// TIA Portal V19 export
FUNCTION "FC90_SentronComm" : Void   // FC90, LAD
{ S7_Optimized_Access := 'TRUE' }
// stored: AutoNumber false, IsIECCheckEnabled true, SetENOAutomatically false
BEGIN

REGION Network 1: Read Sentron Main cabinet
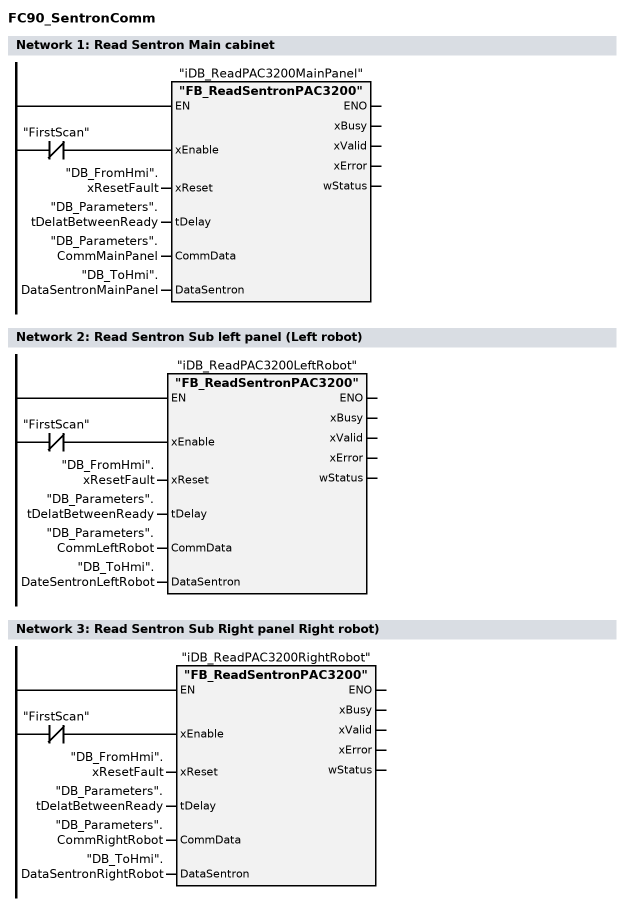
   RUNG wire#powerrail
      "iDB_ReadPAC3200MainPanel"(xEnable := wire#w1, xReset := "DB_FromHmi".xResetFault, tDelay := "DB_Parameters".tDelatBetweenReady, CommData := "DB_Parameters".CommMainPanel, DataSentron := "DB_ToHmi".DataSentronMainPanel, xBusy =>, xValid =>, xError =>, wStatus =>)
   END_RUNG
   RUNG wire#powerrail
      I_Contact( "FirstScan" )
   END_RUNG wire#w1
   // the same network as SCL:
   "iDB_ReadPAC3200MainPanel"(xEnable := NOT "FirstScan",   // "FB_ReadSentronPAC3200"
                           xReset := "DB_FromHmi".xResetFault,
                           tDelay := "DB_Parameters".tDelatBetweenReady,
                           CommData := "DB_Parameters".CommMainPanel,
                           DataSentron := "DB_ToHmi".DataSentronMainPanel);
END_REGION

REGION Network 2: Read Sentron Sub left panel (Left robot)
   RUNG wire#powerrail
      "iDB_ReadPAC3200LeftRobot"(xEnable := wire#w1, xReset := "DB_FromHmi".xResetFault, tDelay := "DB_Parameters".tDelatBetweenReady, CommData := "DB_Parameters".CommLeftRobot, DataSentron := "DB_ToHmi".DateSentronLeftRobot, xBusy =>, xValid =>, xError =>, wStatus =>)
   END_RUNG
   RUNG wire#powerrail
      I_Contact( "FirstScan" )
   END_RUNG wire#w1
   // the same network as SCL:
   "iDB_ReadPAC3200LeftRobot"(xEnable := NOT "FirstScan",   // "FB_ReadSentronPAC3200"
                           xReset := "DB_FromHmi".xResetFault,
                           tDelay := "DB_Parameters".tDelatBetweenReady,
                           CommData := "DB_Parameters".CommLeftRobot,
                           DataSentron := "DB_ToHmi".DateSentronLeftRobot);
END_REGION

REGION Network 3: Read Sentron Sub Right panel Right robot)
   RUNG wire#powerrail
      "iDB_ReadPAC3200RightRobot"(xEnable := wire#w1, xReset := "DB_FromHmi".xResetFault, tDelay := "DB_Parameters".tDelatBetweenReady, CommData := "DB_Parameters".CommRightRobot, DataSentron := "DB_ToHmi".DataSentronRightRobot, xBusy =>, xValid =>, xError =>, wStatus =>)
   END_RUNG
   RUNG wire#powerrail
      I_Contact( "FirstScan" )
   END_RUNG wire#w1
   // the same network as SCL:
   "iDB_ReadPAC3200RightRobot"(xEnable := NOT "FirstScan",   // "FB_ReadSentronPAC3200"
                           xReset := "DB_FromHmi".xResetFault,
                           tDelay := "DB_Parameters".tDelatBetweenReady,
                           CommData := "DB_Parameters".CommRightRobot,
                           DataSentron := "DB_ToHmi".DataSentronRightRobot);
END_REGION
END_FUNCTION
